# EPICS autosave request: iocBoot/iocdelta/auto_settings.req
file hemi_settings.req BL=PINK,DEV=HEMI1
file hemi_settings.req BL=PINK,DEV=HEMI2
file hemi_settings.req BL=PINK,DEV=HEMI3
